# EPICS substitutions: iocBoot/ioc13Keithley_DACpiezo/pid_slow.substitutions
file "$(STD)/stdApp/Db/pid_control.db"
{
pattern
{P,            PID,       INP,           OUT,    LOPR,  HOPR,  DRVL,  DRVH,  PREC,   KP,  KI,   KD,  SCAN}
{13Keithley_DAC_piezo:, PID1,  DMM1Ch8_calc.VAL, DAC1_1,   0,    100,     0,    5,     3,     0.2,  3.,   0.,  ".1 second"}
}
